FUNCTION_BLOCK FB_ExtruderControl

VAR_OUTPUT
	bBusy : BOOL;
	bError : BOOL;
	nErrorId : ERRORID;
END_VAR

VAR_IN_OUT
	pFbExtruderRef : POINTER TO FB_ExtruderRef;
END_VAR

VAR
END_VAR

//Basisklasse

METHOD M_HardStop
VAR_INPUT
END_VAR
END_METHOD

METHOD M_Reset
VAR_INPUT
END_VAR
IF bError THEN
	bError := FALSE;
	nErrorId := 0;
END_IF
END_METHOD

METHOD M_SetCompDistance : ERRORID
VAR_INPUT
	nValue : DINT;
END_VAR
END_METHOD

METHOD M_SetCompFeed : ERRORID
VAR_INPUT
	nValue : DINT;
END_VAR
END_METHOD

METHOD M_SetDistance : ERRORID
VAR_INPUT
	nValue : DINT;
END_VAR
END_METHOD

METHOD M_SetFeed : ERRORID
VAR_INPUT
	nValue : DINT;
END_VAR
END_METHOD

METHOD M_SetRelaxDistance : ERRORID
VAR_INPUT
	nValue : DINT;
END_VAR
END_METHOD

METHOD M_Init
VAR_INPUT
END_VAR
END_METHOD

METHOD M_SetRelaxFeed : ERRORID
VAR_INPUT
	nValue : DINT;
END_VAR
END_METHOD

METHOD M_StartStop
VAR_INPUT
	bStart : BOOL;
END_VAR
END_METHOD

PROPERTY P_nCompDistance : DINT
GET
IF pFbExtruderRef > 0 THEN
	P_nCompDistance := pFbExtruderRef^.P_nCompDistanceOrgin;
END_IF
END_GET
END_PROPERTY

PROPERTY P_nCompFeed : DINT
GET
IF pFbExtruderRef > 0 THEN
	P_nCompFeed := pFbExtruderRef^.P_nCompFeedOrgin; 
END_IF
END_GET
END_PROPERTY

PROPERTY P_nDistance : DINT
GET
IF pFbExtruderRef > 0 THEN
	P_nDistance := pFbExtruderRef^.P_nDistanceOrgin; 
END_IF
END_GET
END_PROPERTY

PROPERTY P_nFeed : DINT
GET
IF pFbExtruderRef > 0 THEN
	P_nFeed := pFbExtruderRef^.P_nFeedOrgin; 
END_IF
END_GET
END_PROPERTY

PROPERTY P_nRelaxDistance : DINT
GET
IF pFbExtruderRef > 0 THEN
	P_nRelaxDistance := pFbExtruderRef^.P_nRelaxDistanceOrgin; 
END_IF
END_GET
END_PROPERTY

PROPERTY P_nRelaxFeed : DINT
GET
IF pFbExtruderRef > 0 THEN
	P_nRelaxFeed := pFbExtruderRef^.P_nRelaxFeedOrgin; 
END_IF
END_GET
END_PROPERTY

END_FUNCTION_BLOCK

(* stored: Version 1.1.0.1, ProductVersion 3.1.4022.7
   POU FB_ExtruderControl: Id {1f5c1974-2d1b-4933-8f2e-3ffa11d6d9fe}, SpecialFunc None
   Method M_HardStop: Id {ce74034e-3c6e-474d-856d-56197108640a}
   Method M_Reset: Id {cd8b4f9a-aa86-4489-937b-2726d865be40}
   Method M_SetCompDistance: Id {cb415c34-3144-4bf0-a8e0-9eba48c0a516}
   Method M_SetCompFeed: Id {265b6c7d-50d7-4a23-97f7-9ed47f3dda46}
   Method M_SetDistance: Id {39ac75e4-39a1-4c59-b5f2-7c19c527fd59}
   Method M_SetFeed: Id {b926a646-5fdd-4746-b071-bdaa5fcd26dc}
   Method M_SetRelaxDistance: Id {06b28c7d-c98b-4679-818e-7664186e4190}
   Method M_Init: Id {26697688-714f-4287-b27a-9f23c99d5872}
   Method M_SetRelaxFeed: Id {b5c1db9a-da29-4ec6-82be-96329ee4fcd5}
   Method M_StartStop: Id {2bd9aed1-bfb2-4975-9e5a-d21407db42ee}
   Property P_nCompDistance: Id {3d802bda-1af6-4b3e-833e-de3fdedb2e9c}
   Get Get: Id {aada73ff-d028-455c-a9b0-e0b91aab6825}
   Property P_nCompFeed: Id {378969a5-f23b-470c-a788-a07178365022}
   Get Get: Id {d046f663-74e7-4137-9d14-7e33f531af75}
   Property P_nDistance: Id {83675b98-e15d-4b1b-8780-69d67a1e8c7e}
   Get Get: Id {ab3c2596-78cc-4777-a2a2-b590724c0fb7}
   Property P_nFeed: Id {45f5e17d-a024-40e8-9630-a736c49ca335}
   Get Get: Id {bb9dedff-bd5d-4bf1-bf5c-3032ac3a61ea}
   Property P_nRelaxDistance: Id {aa5cbfd4-6adb-4e79-84b3-4fd470e682b9}
   Get Get: Id {8e512c5c-e68d-4f82-8373-5ec023e405dc}
   Property P_nRelaxFeed: Id {335f3d6d-0d9c-43c6-b179-d537d4c66bf6}
   Get Get: Id {9272ce5c-6297-4bb2-be7a-4f7aa8bb33fc} *)
